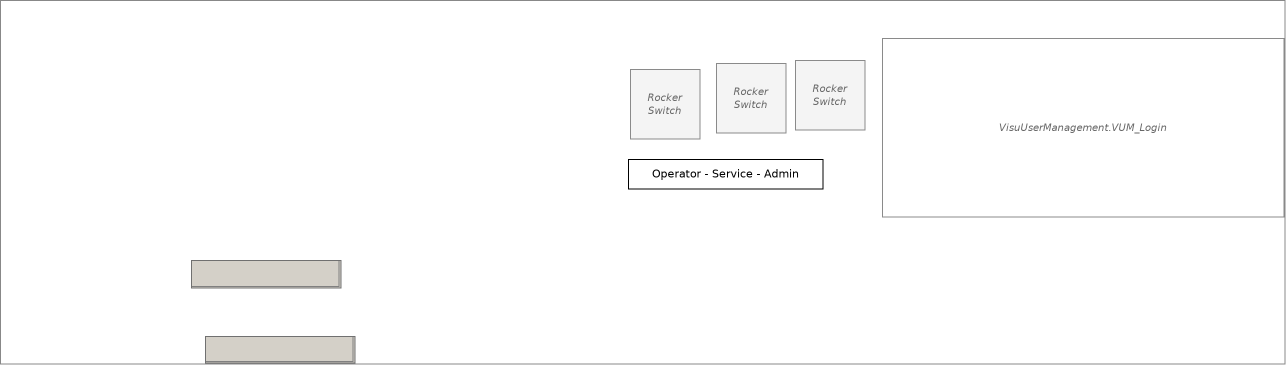
VISUALIZATION Home  // 1286x365
    Rectangle (628,159 195x30), "Operator - Service - Admin"
    Button (205,336 150x27)
        OnMouseClick: VisuUserMgmt Type=Login
    Button (191,260 150x28)
        OnMouseClick: OpenDialog OpenModal=True, OpenCentered=True
    RockerSwitch (630,69 70x70), behaviour: TOGGLE, style: Switch-RockerSwitch-Gray
    RockerSwitch (716,63 70x70), behaviour: TOGGLE, style: Switch-RockerSwitch-Gray
    RockerSwitch (795,60 70x70), behaviour: TOGGLE, style: Switch-RockerSwitch-Gray
    Frame (882,38 402x179)
        shows VisuUserManagement.VUM_Login()
END_VISUALIZATION

(* stored: Version 1.1.0.1, ProductVersion 3.1.4020.6
   Visu Home: Id {b73e9afb-c88e-4dbe-8221-85c1180a67af} *)
